# EPICS substitutions: iocTop/PhaseCavityTiming/PhaseCavityTimingApp/Db/IP330.substitutions
#==============================================================================
#
# Abs:  Acromag IP-330 ADC template
#
# Name: IP330.substitutions
#
#  Auth: 10-Aug-2006, S. Peng         (PENG)
#  Rev:  dd-mmm-yyyy, Reviewer's Name (USERNAME)
#-----------------------------------------------------------------------------
# Mod:
#       dd-mmm-yyyy, First lastname (USERNAME):
#         comment
#
#==============================================================================
#
file IP330.template
{
  # EGU		- Engineering Units
  # EGUF	- Engineering Units Full
  # EGUL	- Engineering Units Low
  # ADEL	- Archive Deadband Limit
  # MDEL	- Monitor Deadband Limit
  # HIHI	- HiHi Alarm Limit
  # HIGH	- High Alarm Limit
  # LOW		- Low  Alarm Limit
  # LOLO	- LoLo Alarm Limit
  pattern { RECORDNAME,          CH, EGUF,  EGUL, ADEL,  MDEL, HIHI,  HIGH, LOW , LOLO,  EGU   }
          { $(CARD):out$(CH), 0,  5.0 ,  0.0 , 0.0 ,  0.0 , 4.5 ,  4.0 , 1.0 , 0.5 ,  Volts }
          { $(CARD):out$(CH), 1,  5.0 ,  0.0 , 0.0 ,  0.0 , 4.5 ,  4.0 , 1.0 , 0.5 ,  Volts }
          { $(CARD):out$(CH), 2,  5.0 ,  0.0 , 0.0 ,  0.0 , 4.5 ,  4.0 , 1.0 , 0.5 ,  Volts }
          { $(CARD):out$(CH), 3,  5.0 ,  0.0 , 0.0 ,  0.0 , 4.5 ,  4.0 , 1.0 , 0.5 ,  Volts }
          { $(CARD):out$(CH), 4,  5.0 ,  0.0 , 0.0 ,  0.0 , 4.5 ,  4.0 , 1.0 , 0.5 ,  Volts }
          { $(CARD):out$(CH), 5,  5.0 ,  0.0 , 0.0 ,  0.0 , 4.5 ,  4.0 , 1.0 , 0.5 ,  Volts }
          { $(CARD):out$(CH), 6,  5.0 ,  0.0 , 0.0 ,  0.0 , 4.5 ,  4.0 , 1.0 , 0.5 ,  Volts }
          { $(CARD):out$(CH), 7,  5.0 ,  0.0 , 0.0 ,  0.0 , 4.5 ,  4.0 , 1.0 , 0.5 ,  Volts }
          { $(CARD):out$(CH), 8,  5.0 ,  0.0 , 0.0 ,  0.0 , 4.5 ,  4.0 , 1.0 , 0.5 ,  Volts }
          { $(CARD):out$(CH), 9,  5.0 ,  0.0 , 0.0 ,  0.0 , 4.5 ,  4.0 , 1.0 , 0.5 ,  Volts }
          { $(CARD):out$(CH), 10, 5.0 ,  0.0 , 0.0 ,  0.0 , 4.5 ,  4.0 , 1.0 , 0.5 ,  Volts }
          { $(CARD):out$(CH), 11, 5.0 ,  0.0 , 0.0 ,  0.0 , 4.5 ,  4.0 , 1.0 , 0.5 ,  Volts }
          { $(CARD):out$(CH), 12, 5.0 ,  0.0 , 0.0 ,  0.0 , 4.5 ,  4.0 , 1.0 , 0.5 ,  Volts }
          { $(CARD):out$(CH), 13, 5.0 ,  0.0 , 0.0 ,  0.0 , 4.5 ,  4.0 , 1.0 , 0.5 ,  Volts }
          { $(CARD):out$(CH), 14, 5.0 ,  0.0 , 0.0 ,  0.0 , 4.5 ,  4.0 , 1.0 , 0.5 ,  Volts }
          { $(CARD):out$(CH), 15, 5.0 ,  0.0 , 0.0 ,  0.0 , 4.5 ,  4.0 , 1.0 , 0.5 ,  Volts }
}
